% RSLogix 500 project PROG.RSS, saved by version 8.30.00.16 %
PROJECT "PROG"    % processor: MicroLogix 1000 %

PROGRAM FILES
  LAD 2   7 rungs
  LAD 3, 4, 5, 6, 7, 8, 9, 10, 11, 12, 13, 14, 15, 16: only END

DATA FILES
  O0 OUTPUT  1 elements
  I1 INPUT  2 elements
  S2 STATUS  33 elements
  B3 BINARY  32 elements
  T4 TIMER  40 elements
  C5 COUNTER  32 elements
  R6 CONTROL  16 elements
  N7 INTEGER  105 elements

LADDER 2
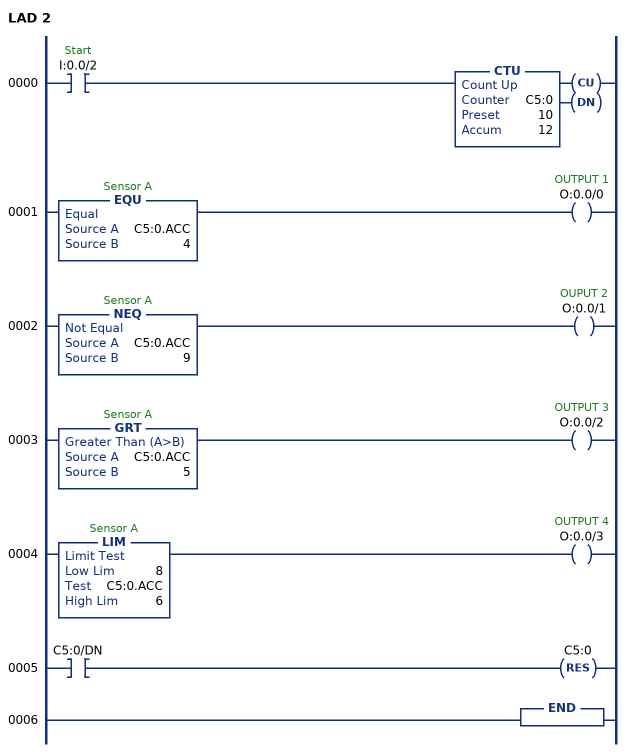
% Rung: 0 %
SOR XIC I:0.0/2 CTU C5:0 10 12 EOR
%   I:0.0/2  "Start" %
% Rung: 1 %
SOR EQU C5:0.ACC 4 OTE O:0.0/0 EOR
%   C5:0.ACC  "Sensor A" %
%   O:0.0/0  "OUTPUT 1" %
% Rung: 2 %
SOR NEQ C5:0.ACC 9 OTE O:0.0/1 EOR
%   C5:0.ACC  "Sensor A" %
%   O:0.0/1  "OUPUT 2" %
% Rung: 3 %
SOR GRT C5:0.ACC 5 OTE O:0.0/2 EOR
%   C5:0.ACC  "Sensor A" %
%   O:0.0/2  "OUTPUT 3" %
% Rung: 4 %
SOR LIM 8 C5:0.ACC 6 OTE O:0.0/3 EOR
%   C5:0.ACC  "Sensor A" %
%   O:0.0/3  "OUTPUT 4" %
% Rung: 5 %
SOR XIC C5:0/DN RES C5:0 EOR
% Rung: 6 %
SOR END EOR

DATA TABLE (non-zero values as saved)
DATA C5
% .PRE .ACC %
% C5:0 % 10 12
